TYPE ST_streamOutputs :
STRUCT
	cycleNo : UDINT;
	on : BOOL;

END_STRUCT
END_TYPE

(* stored: Version 1.1.0.1, ProductVersion 3.1.4024.9
   DUT ST_streamOutputs: Id {6d6a1a82-b3d5-4b08-a46b-082ebaa072b4} *)
